Staubli VAL3: VelocityType.dtx

public num INVALID
public num JOINT
public num BASE_FRAME
public num TOOL_FRAME
